(* Logix 5000 project; controller PLC2_Project_2 Emulate 5570 rev 20.11; software revision 20.00 *)

TASK MainTask (continuous, watchdog 500 ms) : MainProgram

MODULES
   Local : Emulate 5570 (ICP 1, rev 20.11)
      Simulator_Card : vendor 1 type 0 code 15 (ICP 2, rev 1.1, Output RPI 50 ms)
END_MODULES

PROGRAM MainProgram   (* main routine MainRoutine *)
VAR
   Blue_pEye_Delay : TIMER := (PRE := 250);
   Blue_pEye_ONS : BOOL;
   Box_Full : BOOL;
   Box_Full_Delay : TIMER := (PRE := 500);
   Box_InPlace_Delay : TIMER := (PRE := 500);
   Box_InPosition : BOOL;
   Hopper_Interrupt : BOOL;
   I_Switch_BluePhotoEye : BOOL;
   I_Switch_BoxLevelSensor : BOOL;
   I_Switch_BoxProximity : BOOL;
   I_Switch_RedPhotoEye : BOOL;
   Motor_Start_Bit : BOOL;
   Motor_Start_Delay : TIMER := (PRE := 1000);
   Motor_Start_ONS : BOOL;
   Motor_StartStop_Delay : TIMER := (PRE := 500);
   Motor_Stop_Bit : BOOL;
   Motor_Stop_Delay : TIMER := (PRE := 250);
   Motor_Stop_ONS : BOOL;
   O_Hopper_Pecan_En : BOOL;
   O_Hopper_Walnut_En : BOOL;
   O_Motor_En : BOOL;
   PecanBox_Detected : BOOL;
   Red_pEye_Delay : TIMER := (PRE := 250);
   Red_pEye_ONS : BOOL;
   WalnutBox_Detected : BOOL;
END_VAR

ROUTINE Control   (* ladder *)
// Control logic for Hoppers
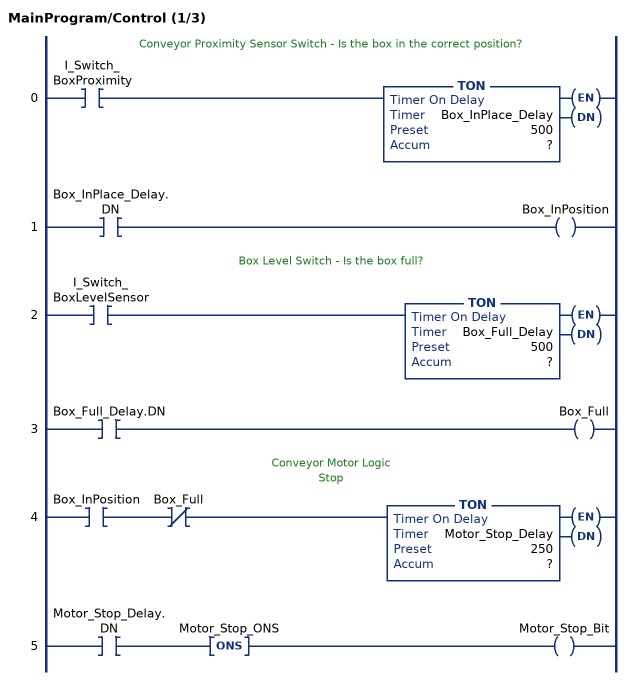
   // Conveyor Proximity Sensor Switch - Is the box in the correct position?
   0: XIC(I_Switch_BoxProximity)TON(Box_InPlace_Delay,?,?);
   1: XIC(Box_InPlace_Delay.DN)OTE(Box_InPosition);
   // Box Level Switch - Is the box full?
   2: XIC(I_Switch_BoxLevelSensor)TON(Box_Full_Delay,?,?);
   3: XIC(Box_Full_Delay.DN)OTE(Box_Full);
   // Conveyor Motor Logic
   // Stop
   4: XIC(Box_InPosition)XIO(Box_Full)TON(Motor_Stop_Delay,?,?);
   5: XIC(Motor_Stop_Delay.DN)ONS(Motor_Stop_ONS)OTE(Motor_Stop_Bit);
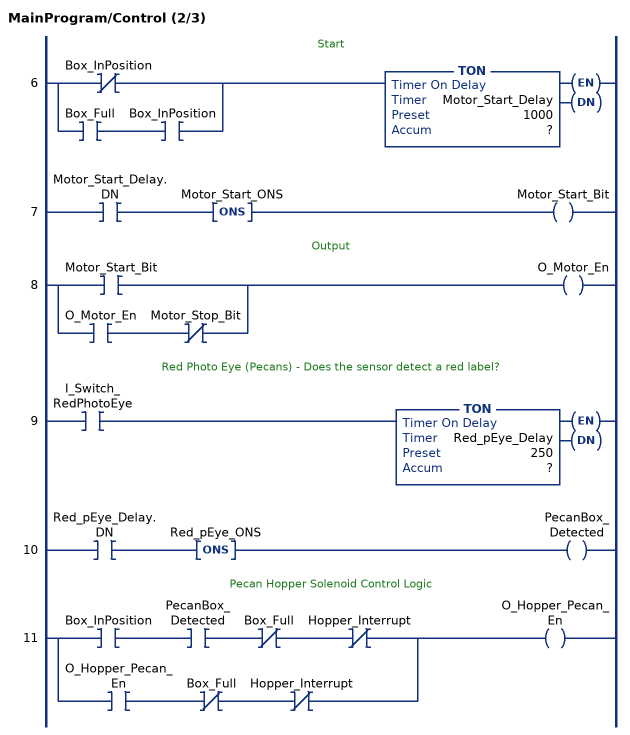
   // Start
   6: [XIO(Box_InPosition) ,XIC(Box_Full) XIC(Box_InPosition) ]TON(Motor_Start_Delay,?,?);
   7: XIC(Motor_Start_Delay.DN)ONS(Motor_Start_ONS)OTE(Motor_Start_Bit);
   // Output
   8: [XIC(Motor_Start_Bit) ,XIC(O_Motor_En) XIO(Motor_Stop_Bit) ]OTE(O_Motor_En);
   // Red Photo Eye (Pecans) - Does the sensor detect a red label?
   9: XIC(I_Switch_RedPhotoEye)TON(Red_pEye_Delay,?,?);
   10: XIC(Red_pEye_Delay.DN)ONS(Red_pEye_ONS)OTE(PecanBox_Detected);
   // Pecan Hopper Solenoid Control Logic
   11: [XIC(Box_InPosition) XIC(PecanBox_Detected) XIO(Box_Full) XIO(Hopper_Interrupt) ,XIC(O_Hopper_Pecan_En) XIO(Box_Full) XIO(Hopper_Interrupt) ]OTE(O_Hopper_Pecan_En);
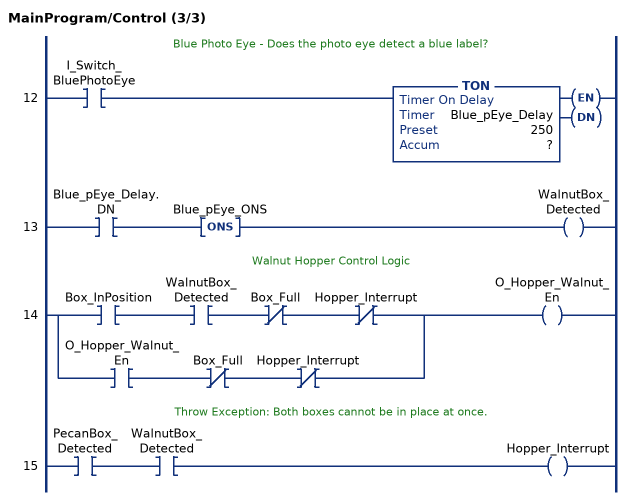
   // Blue Photo Eye - Does the photo eye detect a blue label?
   12: XIC(I_Switch_BluePhotoEye)TON(Blue_pEye_Delay,?,?);
   13: XIC(Blue_pEye_Delay.DN)ONS(Blue_pEye_ONS)OTE(WalnutBox_Detected);
   // Walnut Hopper Control Logic
   14: [XIC(Box_InPosition) XIC(WalnutBox_Detected) XIO(Box_Full) XIO(Hopper_Interrupt) ,XIC(O_Hopper_Walnut_En) XIO(Box_Full) XIO(Hopper_Interrupt) ]OTE(O_Hopper_Walnut_En);
   // Throw Exception: Both boxes cannot be in place at once.
   15: XIC(PecanBox_Detected)XIC(WalnutBox_Detected)OTE(Hopper_Interrupt);
END_ROUTINE

ROUTINE InputOutput   (* ladder *)
// Digital Inputs for Hopper
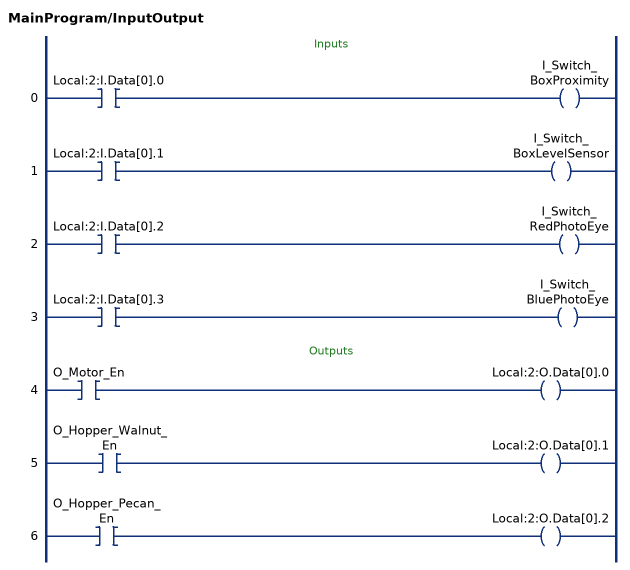
   // Inputs
   0: XIC(Local:2:I.Data[0].0)OTE(I_Switch_BoxProximity);
   1: XIC(Local:2:I.Data[0].1)OTE(I_Switch_BoxLevelSensor);
   2: XIC(Local:2:I.Data[0].2)OTE(I_Switch_RedPhotoEye);
   3: XIC(Local:2:I.Data[0].3)OTE(I_Switch_BluePhotoEye);
   // Outputs
   4: XIC(O_Motor_En)OTE(Local:2:O.Data[0].0);
   5: XIC(O_Hopper_Walnut_En)OTE(Local:2:O.Data[0].1);
   6: XIC(O_Hopper_Pecan_En)OTE(Local:2:O.Data[0].2);
END_ROUTINE

ROUTINE MainRoutine   (* ladder *)
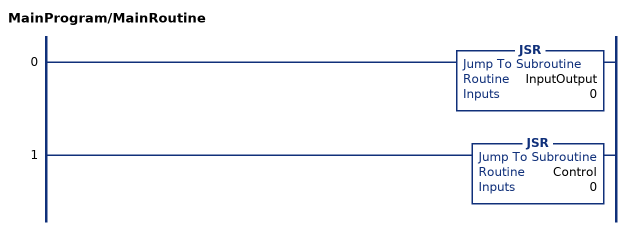
   0: JSR(InputOutput,0);
   1: JSR(Control,0);
END_ROUTINE
END_PROGRAM
